{attribute 'GeneratedUsingTerminal: EL3773-0000-0016'}
{attribute addProperty BoxType "EL3773-0000-0016"}
{attribute addProperty Id "I3_STATUSAT %I*I3_STATUS_B07533568"}
{attribute addProperty CRC "3719215822"}
{attribute addProperty Size "8"}
TYPE L3_Current_Status_DDAEBACE EXTENDS InputBase_8311D824 :
STRUCT
	{attribute addProperty Name "I3_STATUS"}
	I3_STATUS AT %I* : I3_STATUS_B0753356;
END_STRUCT
END_TYPE

(* stored: Version 1.2.0.0, ProductVersion 3.1.4024.11
   DUT L3_Current_Status_DDAEBACE: Id {cead6d9d-2295-447e-b214-c6db7799bf0f} *)
